{attribute 'GeneratedUsingTerminal: IODEVICETYPE_ETHERCATPROT'}
{attribute addProperty BoxType "IODEVICETYPE_ETHERCATPROT"}
{attribute addProperty Id "Term_1_EK1200Term_1_EK1200_E6CF6F51236Term_23_EK1100Term_23_EK1100_046E34D239Term_39_EK1100Term_39_EK1100_42F0B73411SyncUnitsSyncUnits_1397309536InputsInputs_A65FACA410OutputsOutputs_23C0ED1D6InfoDataInfoData_84133AC922"}
{attribute addProperty CRC "3704582866"}
{attribute addProperty Size "360"}
{attribute addProperty Name "Device 1 (EtherCAT)"}
TYPE Device_1_EtherCAT_DCCF72D2 EXTENDS TcoIo.EtcMasterBase_62654B43 :
STRUCT
	{attribute addProperty Name "Term 1 (EK1200)"}
	{attribute addProperty PreviousPort "Device 1 (EtherCAT) : Master"}
	Term_1_EK1200 : Term_1_EK1200_E6CF6F51;
	{attribute addProperty Name "Term 23 (EK1100)"}
	{attribute addProperty PreviousPort "Term 22 (EK1110) : B"}
	Term_23_EK1100 : Term_23_EK1100_046E34D2;
	{attribute addProperty Name "Term 39 (EK1100)"}
	{attribute addProperty PreviousPort "Term 23 (EK1100) : C"}
	Term_39_EK1100 : Term_39_EK1100_42F0B734;
	{attribute addProperty Name "SyncUnits"}
	SyncUnits : SyncUnits_13973095;
	{attribute addProperty Name "Inputs"}
	Inputs : TcoIo.Inputs_A65FACA4;
	{attribute addProperty Name "Outputs"}
	Outputs : TcoIo.Outputs_23C0ED1D;
	{attribute addProperty Name "InfoData"}
	InfoData : TcoIo.InfoData_84133AC9;
END_STRUCT
END_TYPE

(* stored: Version 1.2.0.0, ProductVersion 3.1.4024.11
   DUT Device_1_EtherCAT_DCCF72D2: Id {bc6ee8f5-4552-0e9e-2c8b-90f723e0a8ab} *)
